FUNCTION_BLOCK FACEPLATE (* Controller Faceplate *)
  (* Standard: 61499-1 *)
  (* Version 0.6, 2004-09-08, JHC, Rockwell Automation, Changed CNF to IND. *)
  (* Version 0.5, 2004-09-03, JHC, Rockwell Automation, Changed CNF to IND. *)
  (* Version 0.4, 2004-09-03, JHC, Rockwell Automation, Changed I/O to UINT; added BKGD,COLORS. *)
  (* Version 0.3, 2002-04-25, JHC, Rockwell Automation, Added W, H inputs *)
  (* Version 0.2, 2000-06-20, JHC, Rockwell Automation *)
  (* Version 0.1, 2000-04-29, JHC, Rockwell Automation, SIFB implementation *)
  (* Compiler header: package fb.rt.project; import fb.rt.swing.*; import java.awt.*; *)
  (* Compiler Java Sun JDK 1.4.2 *)
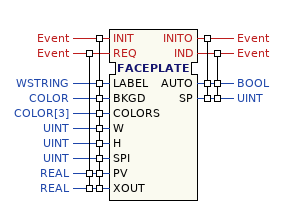
  EVENT_INPUT
    INIT WITH LABEL, W, H, SPI, PV, XOUT, BKGD, COLORS;
    REQ WITH PV, XOUT;
  END_EVENT
  EVENT_OUTPUT
    INITO WITH SP, AUTO;
    IND WITH AUTO, SP; (* Change in AUTO or SP value *)
  END_EVENT
  VAR_INPUT
    LABEL : WSTRING := "   CONTROL FACEPLATE   ";
    BKGD : COLOR := COLOR#lightGray; (* Background color for bars *)
    COLORS : ARRAY [0..2] OF COLOR := [yellow,blue,green]; (* SP,PV,XOUT colors *)
    W : UINT := 20; (* Indicator width *)
    H : UINT := 100; (* Indicator Height *)
    SPI : UINT := 50; (* Initial value for SP, 0-100% *)
    PV : REAL; (* Process Variable, 0-100% *)
    XOUT : REAL; (* Controller Output, 0-100% *)
  END_VAR
  VAR_OUTPUT
    AUTO : BOOL; (* 1=Auto,0=Manual *)
    SP : UINT; (* Set Point, 0-100% *)
  END_VAR
END_FUNCTION_BLOCK
